FUNCTION_BLOCK FB_MSF_Sensor
VAR_INPUT

	bEnable				:	BOOL;
	bRun				: BOOL;
	bInitializedExt	:	BOOL;
	
END_VAR

VAR_OUTPUT
	eStep				:	E_Step;
	eErrStep			:	E_Step;
	nErrId				:	DINT;
	
	bFbEnd				:	BOOL;

	nSlot				:	INT;

	bMotor				:	BOOL;	
END_VAR

VAR_IN_OUT
	stIn		:	ST_CSL_In;
	stParams	: 	ST_CSL_Params;
	stOut		: 	ST_CSL_Out;	
	
END_VAR

VAR
	bInitialized		:	BOOL;
	eNewStep			:	E_Step;
	bEntryAct			:	BOOL;
	fbTonStart			:	TON;
	
	fbMeasure			:	FB_Measuring;
	fbSlot				:	FB_Processing;
	
	
	rPieceValue			:	REAL;
	bEndMeasure			:	BOOL;
	
END_VAR

(*Initialization of the FB_Sensor*)
IF NOT bInitialized OR NOT bInitializedExt THEN
	eNewStep := E_Step.NoStep;
	eStep := E_Step.Stop;
	bEntryAct := FALSE;
	bFbEnd := FALSE;
	bInitialized := TRUE;
ELSE
	
	(*Preamble*)
	
	(*Forcing the Error State*)
	IF NOT bEnable THEN
		eNewStep := E_Step.NeOrError;
	END_IF	
	
	(*State change management*)
	IF eNewStep <> E_Step.NoStep THEN
		eStep := eNewStep;
		eNewStep := E_Step.NoStep;
		bEntryact := FALSE;
	END_IF
	
	(*Filters*)
	fbTonStart(IN := NOT stIn.bPieceSensorInput, PT := T#2S);
		
	(*Case*)
	CASE eStep OF
		(*Stop Step*)
		E_Step.Stop :
			(*Body*)
			bMotor := FALSE;
		
			(*Transition - to Measuring*)
			IF bRun AND bEnable THEN
				eNewStep := E_Step.Start;
			END_IF
			
			(*Exit Act*)
			IF eNewStep <> E_Step.NoStep THEN
				IF eNewStep = E_Step.NeOrError THEN
					eErrStep := eStep;
					//nErrId	:= 16#9999_9999;
				END_IF
			END_IF		
	
		(*Start Step*)
		E_Step.Start :
			(*Body*)
			bMotor := FALSE;
		
			(*Transition - to Measuring*)
			IF fbTonStart.Q AND bEnable THEN
				eNewStep := E_Step.Measuring;
			END_IF
			
			(*Exit Act*)
			IF eNewStep <> E_Step.NoStep THEN
				IF eNewStep = E_Step.NeOrError THEN
					eErrStep := eStep;
					//nErrId	:= 16#9999_9999;
				END_IF
			END_IF
			
		(*Measuring Step*)
		E_Step.Measuring :
			(*Body*)
			bMotor := TRUE;
		
			fbMeasure(Vin := stIn.nColorSensor, Vout := rPieceValue);
			
			(*Transition - to Processing*)
			IF NOT stIn.bPieceSensorOutput AND bEnable THEN
				fbSlot(SensorInput := rPieceValue, stParams := stParams);
				nSlot := fbSlot.slot;
				eNewStep:=E_Step.Stop;
				bInitialized := FALSE;
				bFbEnd := TRUE;
			END_IF
			
			(*Exit Act*)
			IF eNewStep <> E_Step.NoStep THEN
				IF eNewStep = E_Step.NeOrError THEN
					eErrStep := eStep;
					//nErrId	:= 16#9999_9999;
				END_IF
			END_IF
		
		E_Step.NeOrError :
			(*Body*)
			bMotor := FALSE;
		
			bInitialized := FALSE;
			
			(*Exit Act*)
			IF eNewStep <> E_Step.NoStep THEN
				IF eNewStep = E_Step.NeOrError THEN
					eErrStep := eStep;
					//nErrId	:= 16#9999_9999;
				END_IF
			END_IF
			
	END_CASE
END_IF

END_FUNCTION_BLOCK

(* stored: Version 1.1.0.1, ProductVersion 3.1.4024.12
   POU FB_MSF_Sensor: Id {36b94ebf-d3be-44ba-ae1f-96261f197527}, SpecialFunc None *)
